Fanuc KAREL source: wsegtermtype.kl

PROGRAM wsegtermtype
%NOLOCKGROUP
VAR
  p : POSITION
  q : POSITION
  i : INTEGER
  r : REAL
BEGIN
  WITH $SEGTERMTYPE = COARSE MOVE TO p
END wsegtermtype
